FUNCTION_BLOCK FB_Capper IMPLEMENTS IStation
VAR_INPUT
END_VAR
VAR_OUTPUT
END_VAR
VAR
END_VAR

{warning 'add property implementation'}
PROPERTY Busy : BOOL
GET
END_GET
END_PROPERTY

{warning 'add method implementation '}
METHOD Execute : PVOID
END_METHOD

{warning 'add property implementation'}
PROPERTY Faulted : BOOL
GET
END_GET
END_PROPERTY

{warning 'add property implementation'}
PROPERTY Ready : BOOL
GET
END_GET
END_PROPERTY

END_FUNCTION_BLOCK

(* stored: Version 1.1.0.1, ProductVersion 3.1.4024.12
   POU FB_Capper: Id {84003403-a58a-475b-b316-c108bd8518cd}, SpecialFunc None
   Property Busy: Id {e513cc39-182d-4db1-aa76-2ddf2d67e05f}
   Get Get: Id {4c2e7329-e08b-4eb8-bc0e-a9aad6da5bd5}
   Method Execute: Id {3ce6c1cf-617e-4551-9791-e05b0a04d467}
   Property Faulted: Id {27dfba32-5ca0-4c44-bcde-c717b6dba21e}
   Get Get: Id {1653a5f4-852b-43fd-8e37-69fbf6c0d8f8}
   Property Ready: Id {75401c11-93e4-45f6-b582-100bb15a9dd0}
   Get Get: Id {30cab7ee-58fe-4f86-a492-5d86b605ca03} *)
